// TIA Portal V17 export
// export: Created 2023-12-22T15:05:28.3591425Z, ExportSetting WithDefaults, DisplayName Totally Integrated Automation Portal, DisplayVersion V17, DisplayName TIA Portal Openness, DisplayVersion V17, DisplayName TIA Portal Version Control Interface, DisplayVersion V17, DisplayName STEP 7 Professional, DisplayVersion V17, DisplayName STEP 7 Safety, DisplayVersion V17, DisplayName WinCC Advanced, DisplayVersion V17
FUNCTION_BLOCK "DOx_1"   // FB210, LAD
{ S7_Optimized_Access := 'FALSE' }
VERSION : 0.1
// Start - управляющий сигнал из программы
// Q - выходной сигнал контроллера
// pulse - кратность времени в импульсном режиме
// stored: AutoNumber false, IsIECCheckEnabled false, SetENOAutomatically false, UDAEnableTagReadback false
   VAR
      EZ_1_Alarm_Stop { S7_SetPoint := 'True'} : "DO_ex";   // Электролизер 1 (Аварийный останов)
      Red_Signal { S7_SetPoint := 'True'} : "DO_ex";   // Красный сигнал (Колонна)
      KC_1_Start { S7_SetPoint := 'True'} : "DO_ex";   // Промывка фильтра 1 пуск
      KC_2_Start { S7_SetPoint := 'True'} : "DO_ex";   // Промывка фильтра 2 пуск
      command_5 { S7_SetPoint := 'True'} : "DO_ex";
      command_6 { S7_SetPoint := 'True'} : "DO_ex";
      command_7 { S7_SetPoint := 'True'} : "DO_ex";
      command_8 { S7_SetPoint := 'True'} : "DO_ex";
      command_9 { S7_SetPoint := 'True'} : "DO_ex";
      command_10 { S7_SetPoint := 'True'} : "DO_ex";
      command_11 { S7_SetPoint := 'True'} : "DO_ex";
      command_12 { S7_SetPoint := 'True'} : "DO_ex";
   END_VAR
   VAR DB_SPECIFIC
      Time_DTL { S7_SetPoint := 'True'} : DTL;
   END_VAR
   // EZ_1_Alarm_Stop.ADDR_Byte := 0;
   // EZ_1_Alarm_Stop.ADDR_Bit := 1;
   // Red_Signal.ADDR_Bit := 6;
   // KC_1_Start.ADDR_Bit := 4;
   // KC_2_Start.ADDR_Bit := 5;
   VAR_TEMP   // added for the SCL form of the ladder/FBD networks
      _w1 : Bool;
   END_VAR
BEGIN

REGION Network 1
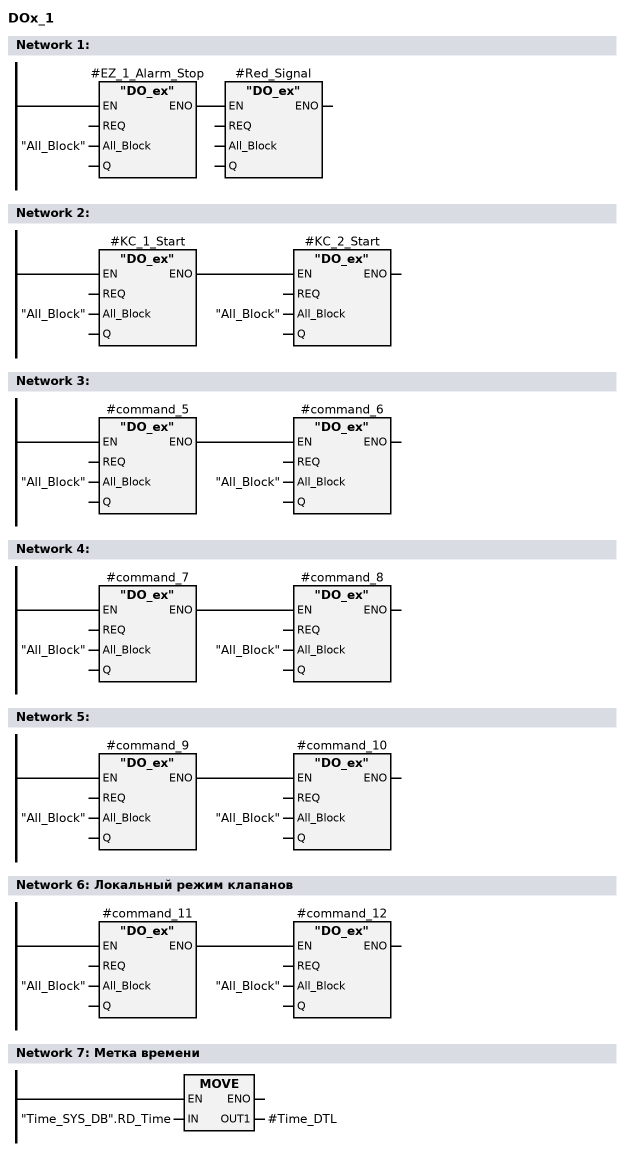
   RUNG wire#powerrail
      #EZ_1_Alarm_Stop(REQ :=, All_Block := "All_Block", Q :=)
      #Red_Signal(REQ :=, All_Block :=, Q :=)
   END_RUNG
   // the same network as SCL:
   #EZ_1_Alarm_Stop(All_Block := "All_Block", ENO => #_w1);   // "DO_ex"
   IF #_w1 THEN
       #Red_Signal();   // "DO_ex"
   END_IF;
END_REGION

REGION Network 2
   RUNG wire#powerrail
      #KC_1_Start(REQ :=, All_Block := "All_Block", Q :=)
      #KC_2_Start(REQ :=, All_Block := "All_Block", Q :=)
   END_RUNG
   // the same network as SCL:
   #KC_1_Start(All_Block := "All_Block", ENO => #_w1);   // "DO_ex"
   IF #_w1 THEN
       #KC_2_Start(All_Block := "All_Block");   // "DO_ex"
   END_IF;
END_REGION

REGION Network 3
   RUNG wire#powerrail
      #command_5(REQ :=, All_Block := "All_Block", Q :=)
      #command_6(REQ :=, All_Block := "All_Block", Q :=)
   END_RUNG
   // the same network as SCL:
   #command_5(All_Block := "All_Block", ENO => #_w1);   // "DO_ex"
   IF #_w1 THEN
       #command_6(All_Block := "All_Block");   // "DO_ex"
   END_IF;
END_REGION

REGION Network 4
   RUNG wire#powerrail
      #command_7(REQ :=, All_Block := "All_Block", Q :=)
      #command_8(REQ :=, All_Block := "All_Block", Q :=)
   END_RUNG
   // the same network as SCL:
   #command_7(All_Block := "All_Block", ENO => #_w1);   // "DO_ex"
   IF #_w1 THEN
       #command_8(All_Block := "All_Block");   // "DO_ex"
   END_IF;
END_REGION

REGION Network 5
   RUNG wire#powerrail
      #command_9(REQ :=, All_Block := "All_Block", Q :=)
      #command_10(REQ :=, All_Block := "All_Block", Q :=)
   END_RUNG
   // the same network as SCL:
   #command_9(All_Block := "All_Block", ENO => #_w1);   // "DO_ex"
   IF #_w1 THEN
       #command_10(All_Block := "All_Block");   // "DO_ex"
   END_IF;
END_REGION

REGION Network 6: Локальный режим клапанов
   RUNG wire#powerrail
      #command_11(REQ :=, All_Block := "All_Block", Q :=)
      #command_12(REQ :=, All_Block := "All_Block", Q :=)
   END_RUNG
   // the same network as SCL:
   #command_11(All_Block := "All_Block", ENO => #_w1);   // "DO_ex"
   IF #_w1 THEN
       #command_12(All_Block := "All_Block");   // "DO_ex"
   END_IF;
END_REGION

REGION Network 7: Метка времени
   RUNG wire#powerrail
      Move(in := "Time_SYS_DB".RD_Time, out1 => #Time_DTL)
   END_RUNG
   // the same network as SCL:
   #Time_DTL := "Time_SYS_DB".RD_Time;
END_REGION
END_FUNCTION_BLOCK
